// TIA Portal project "Numar_random" (V15.1)

(* hardware
DEVICE "S71500/ET200MP station_1"  S7-1500 station
   slot 0: "Rail_0"  Rack  6ES7 590-1***0-0AA0
   slot 1: "PLC_1"  CPU 1513-1 PN  6ES7 513-1AL02-0AB0  V2.6
      slot 3: "CPU display_1"  6ES7591-1AA00-0AA0
DEVICE "HMI_1"  KTP900 Basic PN
   slot 0: "HMI_1"  KTP900 Basic PN  6AV2 123-2JB03-0AX0  15.1.0.0
   slot 1: "HMI_RT_1"  KTP900 Basic PN  6AV2 123-2JB03-0AX0  15.1.0.0
   slot 5: "HMI_1.IE_CP_1"  PROFINET Interface  15.0.1.0
      slot 1: "PROFINET Interface_1"  PROFINET Interface
         slot 1: "Port_1"  Port
*)

// ===== PLC "PLC_1"  CPU 1513-1 PN =====

VAR_GLOBAL   // PLC tag table "Default tag table"
   "System_Byte" AT %MB8069 : Byte;
   "FirstScan" AT %M8069.0 : Bool;
   "DiagStatusUpdate" AT %M8069.1 : Bool;
   "AlwaysTRUE" AT %M8069.2 : Bool;
   "AlwaysFALSE" AT %M8069.3 : Bool;
   "Clock_Byte" AT %MB8080 : Byte;
   "Clock_10Hz" AT %M8080.0 : Bool;
   "Clock_5Hz" AT %M8080.1 : Bool;
   "Clock_2.5Hz" AT %M8080.2 : Bool;
   "Clock_2Hz" AT %M8080.3 : Bool;
   "Clock_1.25Hz" AT %M8080.4 : Bool;
   "Clock_1Hz" AT %M8080.5 : Bool;
   "Clock_0.625Hz" AT %M8080.6 : Bool;
   "Clock_0.5Hz" AT %M8080.7 : Bool;
END_VAR

DATA_BLOCK "Variabile"   // DB1
{ S7_Optimized_Access := 'TRUE' }
VERSION : 0.1
   VAR
      seed : UDInt;
      valoare_returnata : DInt;
      val_min : DInt;
      val_max : DInt;
      valoare_pe_HMI : DInt;
      btn_calculare_nr : Bool;
      btn_reset_avarii : Bool;
      alarma_generala : Bool;
   END_VAR
BEGIN
END_DATA_BLOCK

DATA_BLOCK "Alarme"   // DB2
{ S7_Optimized_Access := 'TRUE' }
VERSION : 0.1
   VAR
      gather : Word;
      "array" : Array[0..15] of Bool;
   END_VAR
BEGIN
END_DATA_BLOCK

FUNCTION "Numar_random" : DInt   // FC1, SCL
{ S7_Optimized_Access := 'TRUE' }
VERSION : 0.1
   VAR_INPUT
      valoare_minima : DInt;
      valoare_maxima : DInt;
      btn_calculeaza_nr : Bool;
   END_VAR
   VAR_IN_OUT
      seed : UDInt;
   END_VAR
   VAR_TEMP
      sysTime : DTL;
      retStatus : Int;
   END_VAR
BEGIN
   IF #seed = 0 THEN
       #retStatus := RD_SYS_T(#sysTime); //pentru posibile erori
       #seed := #sysTime.NANOSECOND; //ia timpul in nanosecunde pentru a calcula mai departe
   END_IF;

   IF #btn_calculeaza_nr THEN
       // Algoritmul de calcul
       #seed := (#seed * 1103515245 + 12345);

       IF #valoare_maxima > #valoare_minima THEN //desi deja am alarma pt asta, un fail safe nu strica
           #Numar_random := #valoare_minima + UDINT_TO_DINT(#seed MOD DINT_TO_UDINT(#valoare_maxima - #valoare_minima));
       ELSE
           #Numar_random := #valoare_minima;
       END_IF;
   ELSE
       //returneza valoarea 0, sa nu se supere compilatorul
       #Numar_random := 0;
   END_IF;
END_FUNCTION

ORGANIZATION_BLOCK "Main"   // OB1, LAD, ProgramCycle
TITLE = "Main Program Sweep (Cycle)"
{ S7_Optimized_Access := 'TRUE' }
VERSION : 0.1
   VAR_INPUT
      Initial_Call : Bool;   // Initial call of this OB
      Remanence : Bool;   // =True, if remanent data are available
   END_VAR
BEGIN

REGION Network 1: gathter de alarme
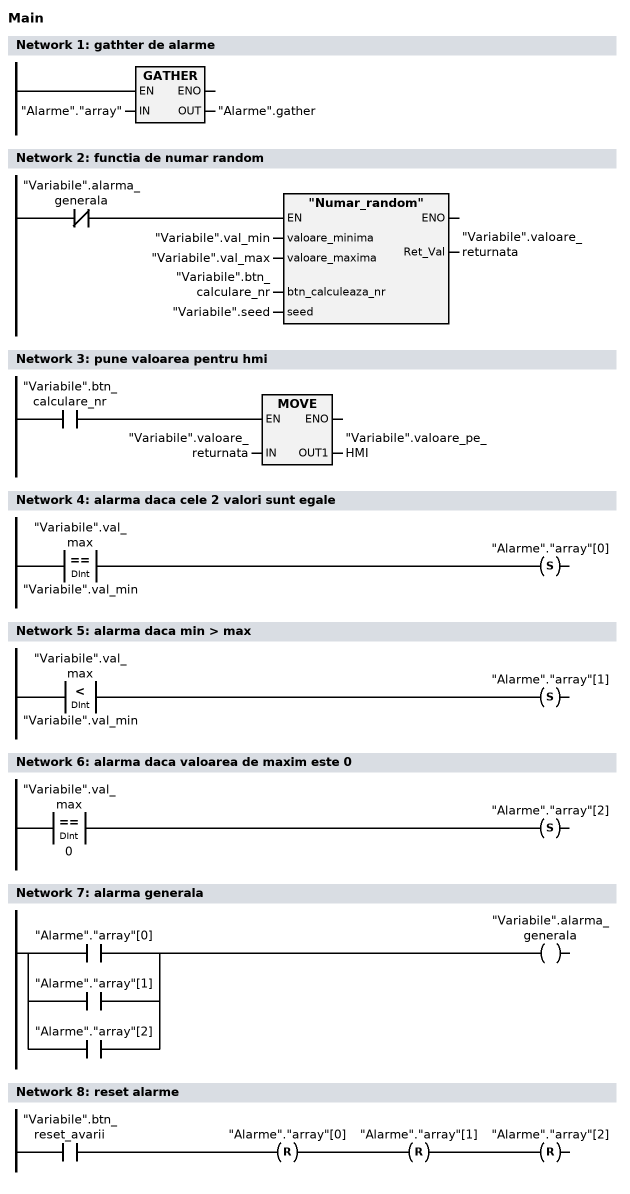
   GATHER(IN := "Alarme"."array", OUT => "Alarme".gather);
END_REGION

REGION Network 2: functia de numar random
   RUNG wire#powerrail
      I_Contact( "Variabile".alarma_generala )
      "Numar_random"(valoare_minima := "Variabile".val_min, valoare_maxima := "Variabile".val_max, btn_calculeaza_nr := "Variabile".btn_calculare_nr, seed := "Variabile".seed, Ret_Val => "Variabile".valoare_returnata)
   END_RUNG
   // the same network as SCL:
   IF NOT "Variabile".alarma_generala THEN
       "Variabile".valoare_returnata := "Numar_random"(valoare_minima := "Variabile".val_min,
                               valoare_maxima := "Variabile".val_max,
                               btn_calculeaza_nr := "Variabile".btn_calculare_nr,
                               seed := "Variabile".seed);
   END_IF;
END_REGION

REGION Network 3: pune valoarea pentru hmi
   RUNG wire#powerrail
      Contact( "Variabile".btn_calculare_nr )
      Move(in := "Variabile".valoare_returnata, out1 => "Variabile".valoare_pe_HMI)
   END_RUNG
   // the same network as SCL:
   IF "Variabile".btn_calculare_nr THEN "Variabile".valoare_pe_HMI := "Variabile".valoare_returnata; END_IF;
END_REGION

REGION Network 4: alarma daca cele 2 valori sunt egale
   RUNG wire#powerrail
      { S7_Templates := "SrcType := DInt" } EQ_Contact(in1 := "Variabile".val_max, in2 := "Variabile".val_min)
      S_Coil( "Alarme"."array"[0] )
   END_RUNG
   // the same network as SCL:
   IF "Variabile".val_max = "Variabile".val_min THEN "Alarme"."array"[0] := TRUE; END_IF;
END_REGION

REGION Network 5: alarma daca min > max
   RUNG wire#powerrail
      { S7_Templates := "SrcType := DInt" } LT_Contact(in1 := "Variabile".val_max, in2 := "Variabile".val_min)
      S_Coil( "Alarme"."array"[1] )
   END_RUNG
   // the same network as SCL:
   IF "Variabile".val_max < "Variabile".val_min THEN "Alarme"."array"[1] := TRUE; END_IF;
END_REGION

REGION Network 6: alarma daca valoarea de maxim este 0
   RUNG wire#powerrail
      { S7_Templates := "SrcType := DInt" } EQ_Contact(in1 := "Variabile".val_max, in2 := 0)
      S_Coil( "Alarme"."array"[2] )
   END_RUNG
   // the same network as SCL:
   IF "Variabile".val_max = 0 THEN "Alarme"."array"[2] := TRUE; END_IF;
END_REGION

REGION Network 7: alarma generala
   RUNG wire#powerrail
      Contact( "Alarme"."array"[0] )
      wire#w1
      Coil( "Variabile".alarma_generala )
   END_RUNG
   RUNG wire#powerrail
      Contact( "Alarme"."array"[1] )
   END_RUNG wire#w1
   RUNG wire#powerrail
      Contact( "Alarme"."array"[2] )
   END_RUNG wire#w1
   // the same network as SCL:
   "Variabile".alarma_generala := "Alarme"."array"[0] OR "Alarme"."array"[1] OR "Alarme"."array"[2];
END_REGION

REGION Network 8: reset alarme
   RUNG wire#powerrail
      Contact( "Variabile".btn_reset_avarii )
      R_Coil( "Alarme"."array"[0] )
      R_Coil( "Alarme"."array"[1] )
      R_Coil( "Alarme"."array"[2] )
   END_RUNG
   // the same network as SCL:
   IF "Variabile".btn_reset_avarii THEN
       "Alarme"."array"[0] := FALSE;
       "Alarme"."array"[1] := FALSE;
       "Alarme"."array"[2] := FALSE;
   END_IF;
END_REGION
END_ORGANIZATION_BLOCK

(* ===== HMI "HMI_RT_1" =====
system functions are stored by id; their names below are inferred from use
connection "HMI_Connection_1": ETHERNET, SMART_S7_1500_OMS

HMI tags "Default tag table"
   "Alarme_gather" : Word = PLC Alarme.gather, 1 s
   "Variabile_valoare_returnata" : DInt = PLC Variabile.valoare_returnata, 1 s
   "Variabile_val_min" : DInt = PLC Variabile.val_min, 1 s
   "Variabile_val_max" : DInt = PLC Variabile.val_max, 1 s
   "Variabile_btn_reset_avarii" : Bool = PLC Variabile.btn_reset_avarii, 1 s
   "Variabile_btn_calculare_nr" : Bool = PLC Variabile.btn_calculare_nr, 1 s
   "Variabile_valoare_pe_HMI" : DInt = PLC Variabile.valoare_pe_HMI, 1 s
   "Variabile_alarma_generala" : Bool = PLC Variabile.alarma_generala, 1 s

discrete alarms
   1: 'Valorile de minim si maxim nu pot sa fie egale', class Errors, trigger "Alarme_gather" bit 0
   2: 'Valoarea de maxim trebuie sa fie mai mare decat cea de minim', class Errors, trigger "Alarme_gather" bit 1
   3: 'Valoarea maxima nu poate sa fie 0', class Errors, trigger "Alarme_gather" bit 2

screen "Main" 800x480, template "Template_1"
   IOField "I/O field_1" at 376,174 size 159x58; FormatPattern 99999
      ProcessValue <- "Variabile_valoare_pe_HMI"
   TextField "Text field_1" at 226,179 size 141x47; Text 'Numar:'
   IOField "I/O field_2" at 652,43 size 96x32; FormatPattern 99999
      ProcessValue <- "Variabile_val_min"
   TextField "Text field_2" at 600,47 size 46x20; Text 'Minim:'
   IOField "I/O field_3" at 652,85 size 96x32; FormatPattern 99999
      ProcessValue <- "Variabile_val_max"
   TextField "Text field_3" at 600,89 size 50x20; Text 'Maxim:'
   Button "Button_1" at 341,262 size 117x55; TextOff 'Genereaza'
      on Release: ResetBit("Variabile_btn_calculare_nr")
      on Press: SetBit("Variabile_btn_calculare_nr")
   Button "Button_2" at 600,135 size 96x32; TextOff 'Reset alarme'
      on Press: SetBit("Variabile_btn_reset_avarii")
      on Release: ResetBit("Variabile_btn_reset_avarii")
   Circle "Circle_1" at 92,64 size 73x73
      Appearance <- "Variabile_alarma_generala"
   TextField "Text field_4" at 72,38 size 112x20; Text 'Alarma generala'
*)